# EPICS substitutions: viocs/si_ps/si_psApp/Db/sfa1.substitutions
file "db/individual.db" {
    pattern { family, pos, num }
        { "SFA1", "01C1", "" }
        { "SFA1", "04C4", "" }
        { "SFA1", "05C1", "" }
        { "SFA1", "08C4", "" }
        { "SFA1", "09C1", "" }
        { "SFA1", "12C4", "" }
        { "SFA1", "13C1", "" }
        { "SFA1", "16C4", "" }
        { "SFA1", "17C1", "" }
        { "SFA1", "20C4", "" }
}
